FUNCTION_BLOCK FB_MotionInterlockStandard IMPLEMENTS I_MotionInterlock
VAR
END_VAR

{warning 'Add method implementation '}
METHOD CanMoveNegative : BOOL
END_METHOD

{warning 'Add method implementation '}
METHOD CanMovePositive : BOOL
END_METHOD

{warning 'Add method implementation '}
METHOD CanPowerOn : BOOL
END_METHOD


METHOD FB_Init: BOOL
VAR_INPUT
    bInitRetains: BOOL; // TRUE: the retain variables are initialized (reset warm / reset cold)
    bInCopyCode: BOOL;  // TRUE: the instance will be copied to the copy code afterward (online change)

    stMotionStage : REFERENCE TO ST_MotionStage;
END_VAR
END_METHOD

END_FUNCTION_BLOCK

(* stored: Version 1.1.0.1
   POU FB_MotionInterlockStandard: Id {31a462b2-5580-4413-95cd-88ebc82053ef}, SpecialFunc None
   Method CanMoveNegative: Id {f56ba45c-32df-4c0f-956e-6c2ae2aaa703}
   Method CanMovePositive: Id {583855e0-9d46-4b87-8aa6-27d6a961238c}
   Method CanPowerOn: Id {fbc62a61-a935-4ef9-9e38-e8705b0d3133}
   Method FB_Init: Id {e78fe736-69b1-4523-b8cc-4361d71b6032} *)
